% RSLogix 500 project Regelventil Zyklussteuerung.RSS, saved by version 8.30.00.16 %
PROJECT "UNTITLED"    % processor: Bul.1763 MicroLogix 1100 Series B %

PROGRAM FILES
  LAD 2 "MAIN"  4 rungs
  LAD 3 "IO"  7 rungs
  LAD 4 "CONTROL"  31 rungs
  LAD 5 "POSITIONS"  6 rungs

DATA FILES
  O0 OUTPUT  4 elements
  I1 INPUT  6 elements
  S2 STATUS  66 elements
  B3 BINARY  4 elements
  T4 TIMER  3 elements
  C5 COUNTER  1 elements
  R6 CONTROL  1 elements
  N7 INTEGER  3 elements
  F8 FLOAT  1 elements

LADDER 2 "MAIN"
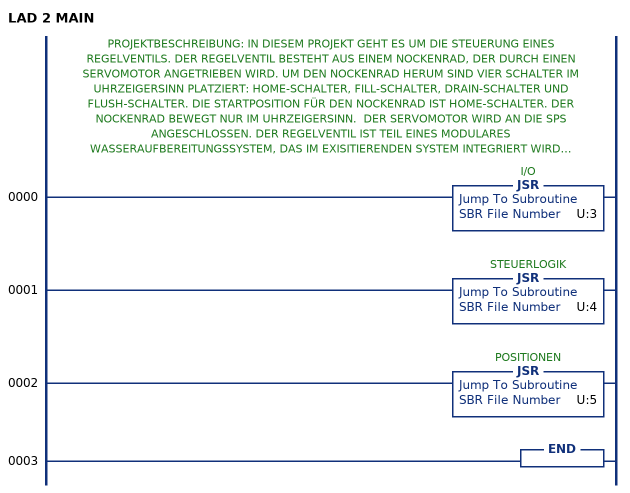
% Rung: 0 %
% PROJEKTBESCHREIBUNG: IN DIESEM PROJEKT GEHT ES UM DIE STEUERUNG EINES REGELVENTILS. DER REGELVENTIL BESTEHT AUS EINEM NOCKENRAD, DER DURCH EINEN SERVOMOTOR ANGETRIEBEN WIRD. UM DEN NOCKENRAD HERUM SIND VIER SCHALTER IM UHRZEIGERSINN PLATZIERT: HOME-SCHALTER, FILL-SCHALTER, DRAIN-SCHALTER UND FLUSH-SCHALTER. DIE STARTPOSITION FÜR DEN NOCKENRAD IST HOME-SCHALTER. DER NOCKENRAD BEWEGT NUR IM UHRZEIGERSINN.  DER SERVOMOTOR WIRD AN DIE SPS ANGESCHLOSSEN. DER REGELVENTIL IST TEIL EINES MODULARES WASSERAUFBEREITUNGSSYSTEM, DAS IM EXISITIERENDEN SYSTEM INTEGRIERT WIRD. DURCH DAS EXISTIERENDE SYSTEM KANN EIN ZYKLUSBEFEHL ERFOLGEN. ANHAND DIESES BEFEHLS WIRD EIN ZYKLUS DURCHGEFÜHRT. DER ZYKLUS DURCHLÄUFT FOLGENDE SCHRITTE:
% 1) FALLS NOCKENRAD SICH NICHT AN STARTPOSITION BEFINDET(HOME-SCHALTER NICHT EINGESCHALTET), DREHT DER NOCKENRAD BIS DER HOME-SCHALTER EINGESCHLATET IST:
% 2) DANN BEWEGT SICH DER NOCKENRAD BIS DER FILL-SCHALTER EINGESCHALTET IST UND DER FILLVORGANG WIRD FÜR 10 SEKUNDEN DURCHGEFÜHRT.
% 3) NACH 10 SEKUNDEN,DER NOCKENRAD BEWEGT SICH WEITER  BIS DER DRAIN-SCHALTER EINGESCHALTET IST. DER DRAINVORGANG WIRD FÜR 20 SEKUNDEN DURCHGEFÜHRT.
% 4) NACH 20 SEKUNDEN, DER NOCKENRAD BEWEGT SICH WEITER BIS DER FLUSH-SCHALTET EINGESCHALTET IST. DER FLUSHVORGAGN WIRD FÜR 10 SEKUNDEN DURCHGEFÜHRT.
% 5) NACH 10 SEKUNDEN, DER NOCKENRAD DREHT SICH WEITER BIS DER HOME-SCHALTET WIEDER EINSCHALTET WIRD. DER ZYKLUS KOMMT ZUM ENDE.
% FERNER HAT DAS PROGRAM DAS INTERRUPT-BIT B3:0/0. FALLS SIE AKTIV WIRD UND DER REGELVENTIL DEN ZYKLUS DURCHLÄUFT, WIRD DER ZYKLUS UNTERBROCHEN UND DER REGELVENTIL KOMMT ZUR STARTPOSITION: %
SOR JSR U:3 EOR
%   U:3  "I/O" %
% Rung: 1 %
SOR JSR U:4 EOR
%   U:4  "STEUERLOGIK" %
% Rung: 2 %
SOR JSR U:5 EOR
%   U:5  "POSITIONEN" %
% Rung: 3 %
SOR END EOR

LADDER 3 "IO"
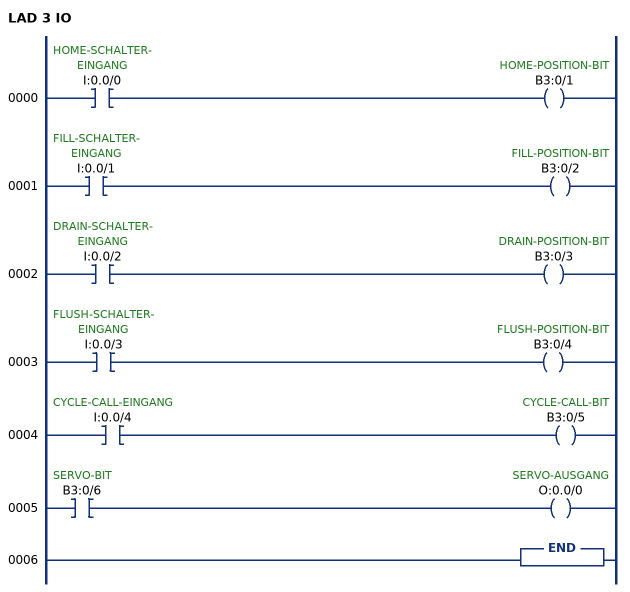
% Rung: 0 %
SOR XIC I:0.0/0 OTE B3:0/1 EOR
%   I:0.0/0  "HOME-SCHALTER- EINGANG" %
%   B3:0/1  "HOME-POSITION-BIT" %
% Rung: 1 %
SOR XIC I:0.0/1 OTE B3:0/2 EOR
%   I:0.0/1  "FILL-SCHALTER- EINGANG" %
%   B3:0/2  "FILL-POSITION-BIT" %
% Rung: 2 %
SOR XIC I:0.0/2 OTE B3:0/3 EOR
%   I:0.0/2  "DRAIN-SCHALTER- EINGANG" %
%   B3:0/3  "DRAIN-POSITION-BIT" %
% Rung: 3 %
SOR XIC I:0.0/3 OTE B3:0/4 EOR
%   I:0.0/3  "FLUSH-SCHALTER- EINGANG" %
%   B3:0/4  "FLUSH-POSITION-BIT" %
% Rung: 4 %
SOR XIC I:0.0/4 OTE B3:0/5 EOR
%   I:0.0/4  "CYCLE-CALL-EINGANG" %
%   B3:0/5  "CYCLE-CALL-BIT" %
% Rung: 5 %
SOR XIC B3:0/6 OTE O:0.0/0 EOR
%   B3:0/6  "SERVO-BIT" %
%   O:0.0/0  "SERVO-AUSGANG" %
% Rung: 6 %
SOR END EOR

LADDER 4 "CONTROL"
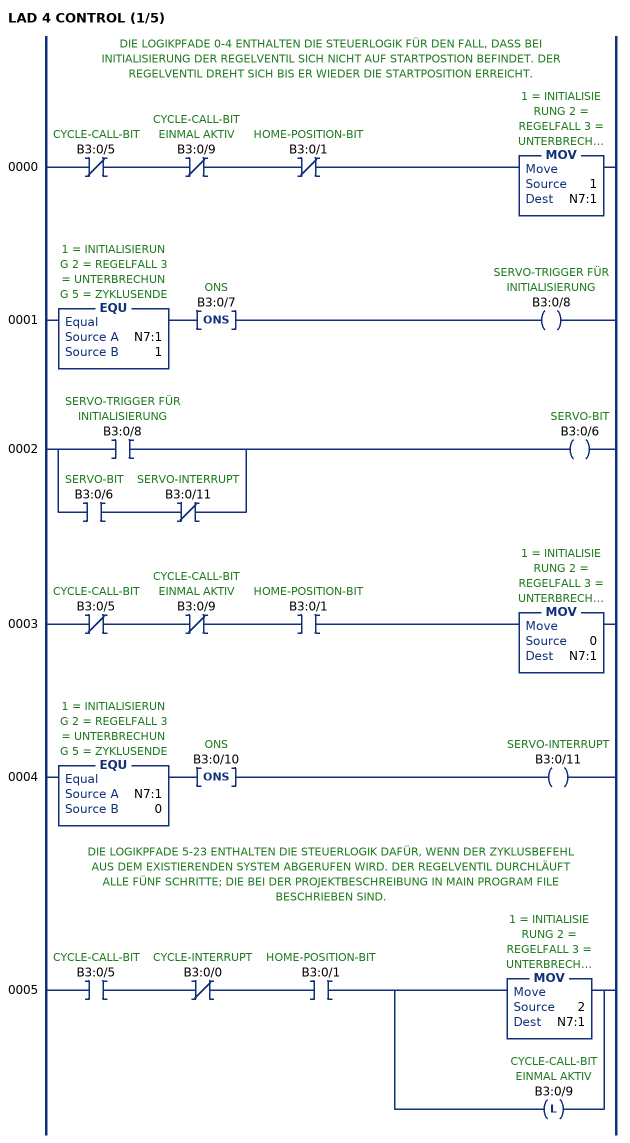
% Rung: 0 %  % edit flag set %
% DIE LOGIKPFADE 0-4 ENTHALTEN DIE STEUERLOGIK FÜR DEN FALL, DASS BEI INITIALISIERUNG DER REGELVENTIL SICH NICHT AUF STARTPOSTION BEFINDET. DER REGELVENTIL DREHT SICH BIS ER WIEDER DIE STARTPOSITION ERREICHT. %
SOR XIO B3:0/5 XIO B3:0/9 XIO B3:0/1 MOV 1 N7:1 EOR
%   B3:0/5  "CYCLE-CALL-BIT" %
%   B3:0/9  "CYCLE-CALL-BIT EINMAL AKTIV" %
%   B3:0/1  "HOME-POSITION-BIT" %
%   N7:1  "1 = INITIALISIERUNG 2 = REGELFALL 3 = UNTERBRECHUNG 5 = ZYKLUSENDE" %
% Rung: 1 %
SOR EQU N7:1 1 ONS B3:0/7 OTE B3:0/8 EOR
%   N7:1  "1 = INITIALISIERUNG 2 = REGELFALL 3 = UNTERBRECHUNG 5 = ZYKLUSENDE" %
%   B3:0/7  "ONS" %
%   B3:0/8  "SERVO-TRIGGER FÜR INITIALISIERUNG" %
% Rung: 2 %
SOR BST XIC B3:0/8 NXB XIC B3:0/6 XIO B3:0/11 BND OTE B3:0/6 EOR
%   B3:0/8  "SERVO-TRIGGER FÜR INITIALISIERUNG" %
%   B3:0/6  "SERVO-BIT" %
%   B3:0/11  "SERVO-INTERRUPT" %
% Rung: 3 %
SOR XIO B3:0/5 XIO B3:0/9 XIC B3:0/1 MOV 0 N7:1 EOR
%   B3:0/5  "CYCLE-CALL-BIT" %
%   B3:0/9  "CYCLE-CALL-BIT EINMAL AKTIV" %
%   B3:0/1  "HOME-POSITION-BIT" %
%   N7:1  "1 = INITIALISIERUNG 2 = REGELFALL 3 = UNTERBRECHUNG 5 = ZYKLUSENDE" %
% Rung: 4 %
SOR EQU N7:1 0 ONS B3:0/10 OTE B3:0/11 EOR
%   N7:1  "1 = INITIALISIERUNG 2 = REGELFALL 3 = UNTERBRECHUNG 5 = ZYKLUSENDE" %
%   B3:0/10  "ONS" %
%   B3:0/11  "SERVO-INTERRUPT" %
% Rung: 5 %
% DIE LOGIKPFADE 5-23 ENTHALTEN DIE STEUERLOGIK DAFÜR, WENN DER ZYKLUSBEFEHL AUS DEM EXISTIERENDEN SYSTEM ABGERUFEN WIRD. DER REGELVENTIL DURCHLÄUFT  ALLE FÜNF SCHRITTE; DIE BEI DER PROJEKTBESCHREIBUNG IN MAIN PROGRAM FILE BESCHRIEBEN SIND. %
SOR XIC B3:0/5 XIO B3:0/0 XIC B3:0/1 BST MOV 2 N7:1 NXB OTL B3:0/9 BND EOR
%   B3:0/5  "CYCLE-CALL-BIT" %
%   B3:0/0  "CYCLE-INTERRUPT" %
%   B3:0/1  "HOME-POSITION-BIT" %
%   N7:1  "1 = INITIALISIERUNG 2 = REGELFALL 3 = UNTERBRECHUNG 5 = ZYKLUSENDE" %
%   B3:0/9  "CYCLE-CALL-BIT EINMAL AKTIV" %

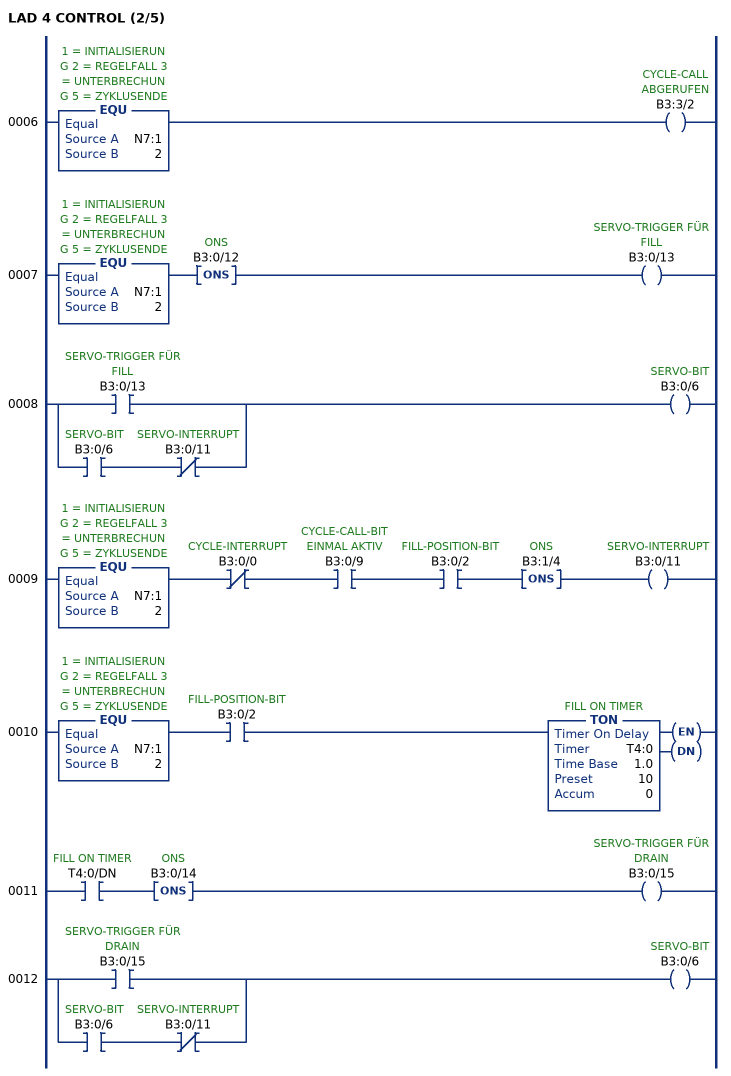
% Rung: 6 %
SOR EQU N7:1 2 OTE B3:3/2 EOR
%   N7:1  "1 = INITIALISIERUNG 2 = REGELFALL 3 = UNTERBRECHUNG 5 = ZYKLUSENDE" %
%   B3:3/2  "CYCLE-CALL ABGERUFEN" %
% Rung: 7 %
SOR EQU N7:1 2 ONS B3:0/12 OTE B3:0/13 EOR
%   N7:1  "1 = INITIALISIERUNG 2 = REGELFALL 3 = UNTERBRECHUNG 5 = ZYKLUSENDE" %
%   B3:0/12  "ONS" %
%   B3:0/13  "SERVO-TRIGGER FÜR FILL" %
% Rung: 8 %
SOR BST XIC B3:0/13 NXB XIC B3:0/6 XIO B3:0/11 BND OTE B3:0/6 EOR
%   B3:0/13  "SERVO-TRIGGER FÜR FILL" %
%   B3:0/6  "SERVO-BIT" %
%   B3:0/11  "SERVO-INTERRUPT" %
% Rung: 9 %
SOR EQU N7:1 2 XIO B3:0/0 XIC B3:0/9 XIC B3:0/2 ONS B3:1/4 OTE B3:0/11 EOR
%   N7:1  "1 = INITIALISIERUNG 2 = REGELFALL 3 = UNTERBRECHUNG 5 = ZYKLUSENDE" %
%   B3:0/0  "CYCLE-INTERRUPT" %
%   B3:0/9  "CYCLE-CALL-BIT EINMAL AKTIV" %
%   B3:0/2  "FILL-POSITION-BIT" %
%   B3:1/4  "ONS" %
%   B3:0/11  "SERVO-INTERRUPT" %
% Rung: 10 %
SOR EQU N7:1 2 XIC B3:0/2 TON T4:0 1.0 10 0 EOR
%   N7:1  "1 = INITIALISIERUNG 2 = REGELFALL 3 = UNTERBRECHUNG 5 = ZYKLUSENDE" %
%   B3:0/2  "FILL-POSITION-BIT" %
%   T4:0  "FILL ON TIMER" %
% Rung: 11 %
SOR XIC T4:0/DN ONS B3:0/14 OTE B3:0/15 EOR
%   T4:0  "FILL ON TIMER" %
%   B3:0/14  "ONS" %
%   B3:0/15  "SERVO-TRIGGER FÜR DRAIN" %
% Rung: 12 %
SOR BST XIC B3:0/15 NXB XIC B3:0/6 XIO B3:0/11 BND OTE B3:0/6 EOR
%   B3:0/15  "SERVO-TRIGGER FÜR DRAIN" %
%   B3:0/6  "SERVO-BIT" %
%   B3:0/11  "SERVO-INTERRUPT" %

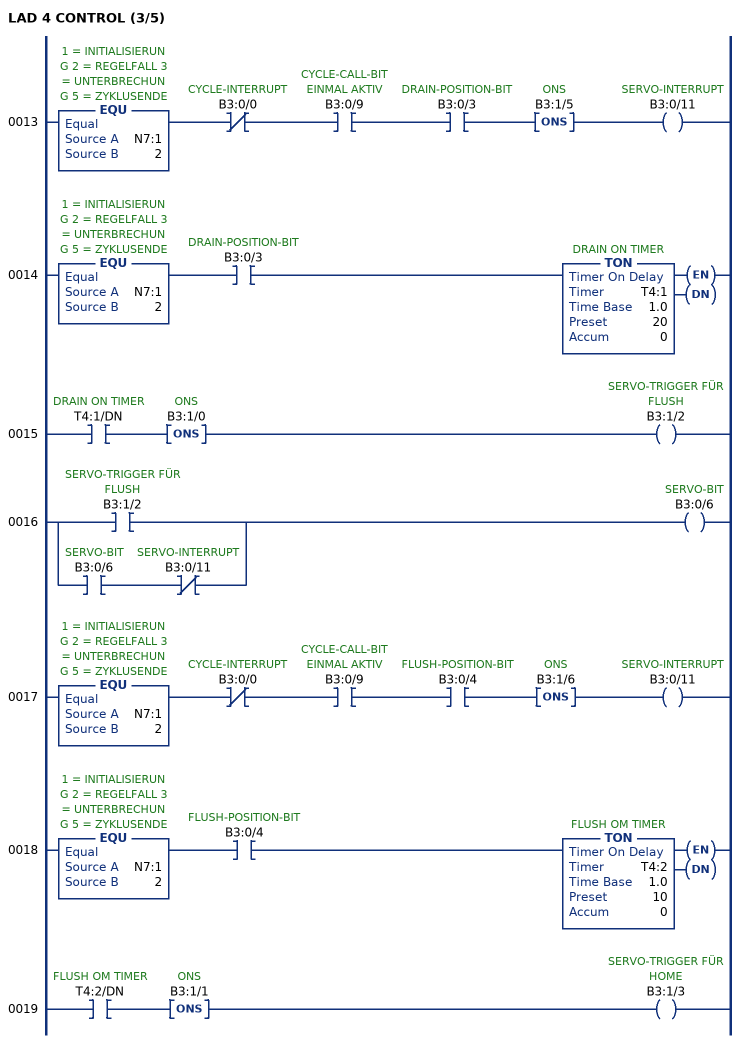
% Rung: 13 %
SOR EQU N7:1 2 XIO B3:0/0 XIC B3:0/9 XIC B3:0/3 ONS B3:1/5 OTE B3:0/11 EOR
%   N7:1  "1 = INITIALISIERUNG 2 = REGELFALL 3 = UNTERBRECHUNG 5 = ZYKLUSENDE" %
%   B3:0/0  "CYCLE-INTERRUPT" %
%   B3:0/9  "CYCLE-CALL-BIT EINMAL AKTIV" %
%   B3:0/3  "DRAIN-POSITION-BIT" %
%   B3:1/5  "ONS" %
%   B3:0/11  "SERVO-INTERRUPT" %
% Rung: 14 %
SOR EQU N7:1 2 XIC B3:0/3 TON T4:1 1.0 20 0 EOR
%   N7:1  "1 = INITIALISIERUNG 2 = REGELFALL 3 = UNTERBRECHUNG 5 = ZYKLUSENDE" %
%   B3:0/3  "DRAIN-POSITION-BIT" %
%   T4:1  "DRAIN ON TIMER" %
% Rung: 15 %
SOR XIC T4:1/DN ONS B3:1/0 OTE B3:1/2 EOR
%   T4:1  "DRAIN ON TIMER" %
%   B3:1/0  "ONS" %
%   B3:1/2  "SERVO-TRIGGER FÜR FLUSH" %
% Rung: 16 %
SOR BST XIC B3:1/2 NXB XIC B3:0/6 XIO B3:0/11 BND OTE B3:0/6 EOR
%   B3:1/2  "SERVO-TRIGGER FÜR FLUSH" %
%   B3:0/6  "SERVO-BIT" %
%   B3:0/11  "SERVO-INTERRUPT" %
% Rung: 17 %
SOR EQU N7:1 2 XIO B3:0/0 XIC B3:0/9 XIC B3:0/4 ONS B3:1/6 OTE B3:0/11 EOR
%   N7:1  "1 = INITIALISIERUNG 2 = REGELFALL 3 = UNTERBRECHUNG 5 = ZYKLUSENDE" %
%   B3:0/0  "CYCLE-INTERRUPT" %
%   B3:0/9  "CYCLE-CALL-BIT EINMAL AKTIV" %
%   B3:0/4  "FLUSH-POSITION-BIT" %
%   B3:1/6  "ONS" %
%   B3:0/11  "SERVO-INTERRUPT" %
% Rung: 18 %
SOR EQU N7:1 2 XIC B3:0/4 TON T4:2 1.0 10 0 EOR
%   N7:1  "1 = INITIALISIERUNG 2 = REGELFALL 3 = UNTERBRECHUNG 5 = ZYKLUSENDE" %
%   B3:0/4  "FLUSH-POSITION-BIT" %
%   T4:2  "FLUSH OM TIMER" %
% Rung: 19 %
SOR XIC T4:2/DN ONS B3:1/1 OTE B3:1/3 EOR
%   T4:2  "FLUSH OM TIMER" %
%   B3:1/1  "ONS" %
%   B3:1/3  "SERVO-TRIGGER FÜR HOME" %

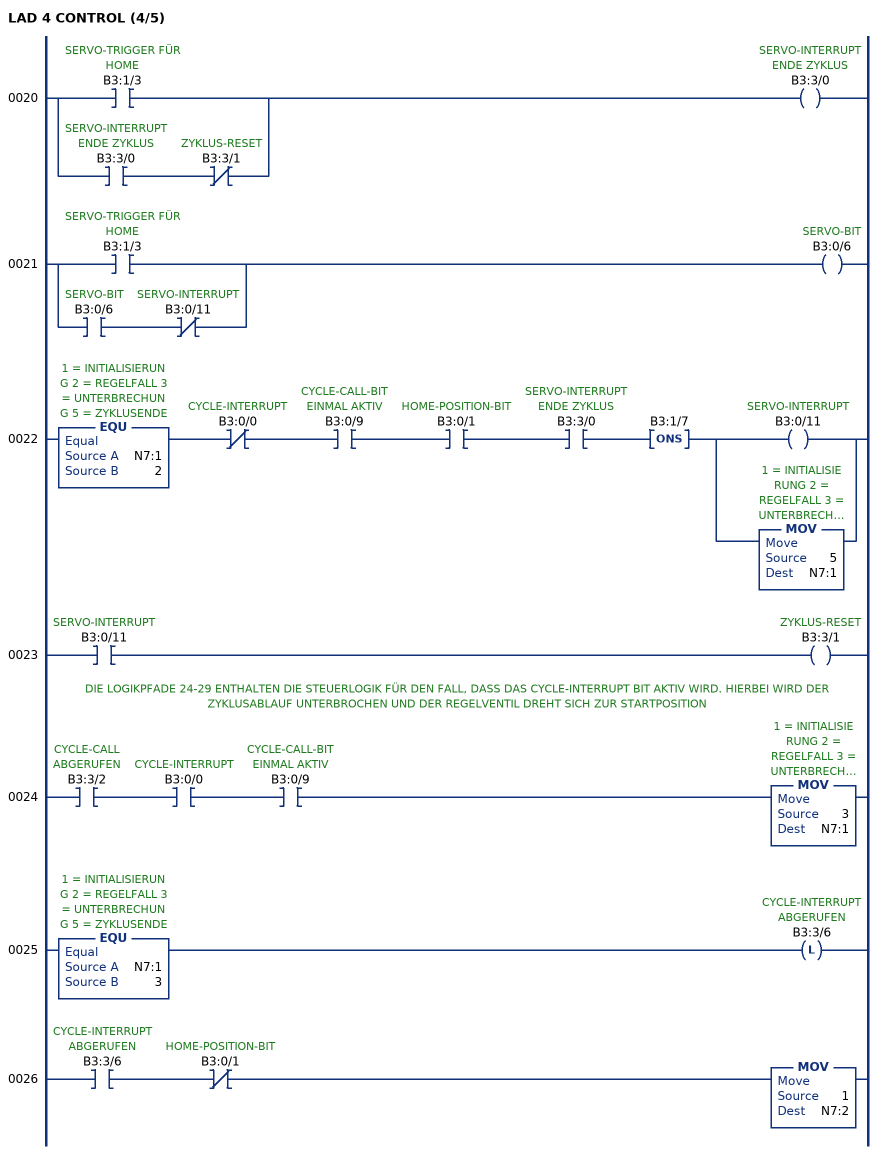
% Rung: 20 %
SOR BST XIC B3:1/3 NXB XIC B3:3/0 XIO B3:3/1 BND OTE B3:3/0 EOR
%   B3:1/3  "SERVO-TRIGGER FÜR HOME" %
%   B3:3/0  "SERVO-INTERRUPT ENDE ZYKLUS" %
%   B3:3/1  "ZYKLUS-RESET" %
% Rung: 21 %
SOR BST XIC B3:1/3 NXB XIC B3:0/6 XIO B3:0/11 BND OTE B3:0/6 EOR
%   B3:1/3  "SERVO-TRIGGER FÜR HOME" %
%   B3:0/6  "SERVO-BIT" %
%   B3:0/11  "SERVO-INTERRUPT" %
% Rung: 22 %
SOR EQU N7:1 2 XIO B3:0/0 XIC B3:0/9 XIC B3:0/1 XIC B3:3/0 ONS B3:1/7 BST OTE B3:0/11 NXB MOV 5 N7:1 BND EOR
%   N7:1  "1 = INITIALISIERUNG 2 = REGELFALL 3 = UNTERBRECHUNG 5 = ZYKLUSENDE" %
%   B3:0/0  "CYCLE-INTERRUPT" %
%   B3:0/9  "CYCLE-CALL-BIT EINMAL AKTIV" %
%   B3:0/1  "HOME-POSITION-BIT" %
%   B3:3/0  "SERVO-INTERRUPT ENDE ZYKLUS" %
%   B3:0/11  "SERVO-INTERRUPT" %
% Rung: 23 %
SOR XIC B3:0/11 OTE B3:3/1 EOR
%   B3:0/11  "SERVO-INTERRUPT" %
%   B3:3/1  "ZYKLUS-RESET" %
% Rung: 24 %
% DIE LOGIKPFADE 24-29 ENTHALTEN DIE STEUERLOGIK FÜR DEN FALL, DASS DAS CYCLE-INTERRUPT BIT AKTIV WIRD. HIERBEI WIRD DER ZYKLUSABLAUF UNTERBROCHEN UND DER REGELVENTIL DREHT SICH ZUR STARTPOSITION %
SOR XIC B3:3/2 XIC B3:0/0 XIC B3:0/9 MOV 3 N7:1 EOR
%   B3:3/2  "CYCLE-CALL ABGERUFEN" %
%   B3:0/0  "CYCLE-INTERRUPT" %
%   B3:0/9  "CYCLE-CALL-BIT EINMAL AKTIV" %
%   N7:1  "1 = INITIALISIERUNG 2 = REGELFALL 3 = UNTERBRECHUNG 5 = ZYKLUSENDE" %
% Rung: 25 %
SOR EQU N7:1 3 OTL B3:3/6 EOR
%   N7:1  "1 = INITIALISIERUNG 2 = REGELFALL 3 = UNTERBRECHUNG 5 = ZYKLUSENDE" %
%   B3:3/6  "CYCLE-INTERRUPT ABGERUFEN" %
% Rung: 26 %
SOR XIC B3:3/6 XIO B3:0/1 MOV 1 N7:2 EOR
%   B3:3/6  "CYCLE-INTERRUPT ABGERUFEN" %
%   B3:0/1  "HOME-POSITION-BIT" %

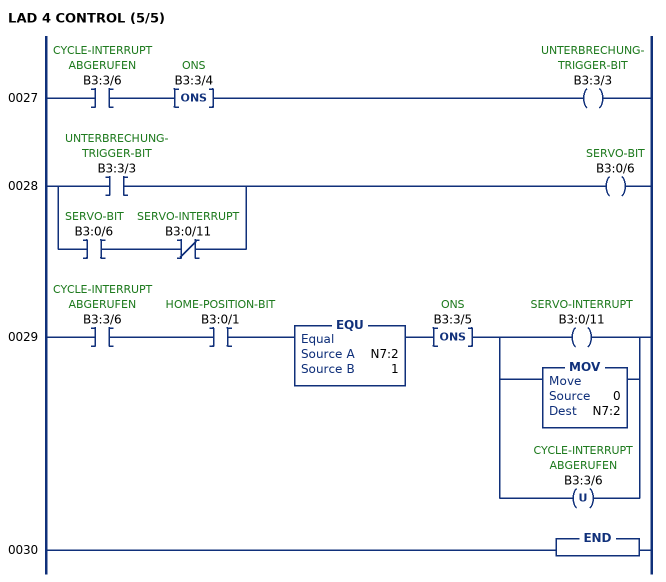
% Rung: 27 %
SOR XIC B3:3/6 ONS B3:3/4 OTE B3:3/3 EOR
%   B3:3/6  "CYCLE-INTERRUPT ABGERUFEN" %
%   B3:3/4  "ONS" %
%   B3:3/3  "UNTERBRECHUNG- TRIGGER-BIT" %
% Rung: 28 %
SOR BST XIC B3:3/3 NXB XIC B3:0/6 XIO B3:0/11 BND OTE B3:0/6 EOR
%   B3:3/3  "UNTERBRECHUNG- TRIGGER-BIT" %
%   B3:0/6  "SERVO-BIT" %
%   B3:0/11  "SERVO-INTERRUPT" %
% Rung: 29 %
SOR XIC B3:3/6 XIC B3:0/1 EQU N7:2 1 ONS B3:3/5 BST OTE B3:0/11 NXB MOV 0 N7:2 NXB OTU B3:3/6 BND EOR
%   B3:3/6  "CYCLE-INTERRUPT ABGERUFEN" %
%   B3:0/1  "HOME-POSITION-BIT" %
%   B3:3/5  "ONS" %
%   B3:0/11  "SERVO-INTERRUPT" %
% Rung: 30 %
SOR END EOR

LADDER 5 "POSITIONS"
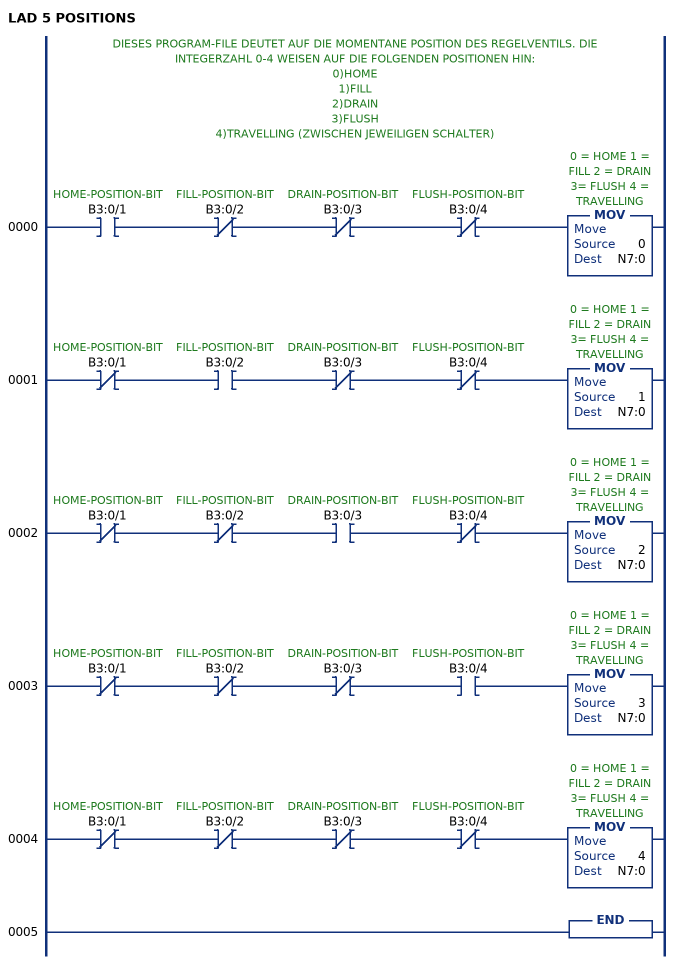
% Rung: 0 %
% DIESES PROGRAM-FILE DEUTET AUF DIE MOMENTANE POSITION DES REGELVENTILS. DIE INTEGERZAHL 0-4 WEISEN AUF DIE FOLGENDEN POSITIONEN HIN:
% 0)HOME
% 1)FILL
% 2)DRAIN
% 3)FLUSH
% 4)TRAVELLING (ZWISCHEN JEWEILIGEN SCHALTER) %
SOR XIC B3:0/1 XIO B3:0/2 XIO B3:0/3 XIO B3:0/4 MOV 0 N7:0 EOR
%   B3:0/1  "HOME-POSITION-BIT" %
%   B3:0/2  "FILL-POSITION-BIT" %
%   B3:0/3  "DRAIN-POSITION-BIT" %
%   B3:0/4  "FLUSH-POSITION-BIT" %
%   N7:0  "0 = HOME 1 = FILL 2 = DRAIN 3= FLUSH 4 = TRAVELLING" %
% Rung: 1 %
SOR XIO B3:0/1 XIC B3:0/2 XIO B3:0/3 XIO B3:0/4 MOV 1 N7:0 EOR
%   B3:0/1  "HOME-POSITION-BIT" %
%   B3:0/2  "FILL-POSITION-BIT" %
%   B3:0/3  "DRAIN-POSITION-BIT" %
%   B3:0/4  "FLUSH-POSITION-BIT" %
%   N7:0  "0 = HOME 1 = FILL 2 = DRAIN 3= FLUSH 4 = TRAVELLING" %
% Rung: 2 %
SOR XIO B3:0/1 XIO B3:0/2 XIC B3:0/3 XIO B3:0/4 MOV 2 N7:0 EOR
%   B3:0/1  "HOME-POSITION-BIT" %
%   B3:0/2  "FILL-POSITION-BIT" %
%   B3:0/3  "DRAIN-POSITION-BIT" %
%   B3:0/4  "FLUSH-POSITION-BIT" %
%   N7:0  "0 = HOME 1 = FILL 2 = DRAIN 3= FLUSH 4 = TRAVELLING" %
% Rung: 3 %
SOR XIO B3:0/1 XIO B3:0/2 XIO B3:0/3 XIC B3:0/4 MOV 3 N7:0 EOR
%   B3:0/1  "HOME-POSITION-BIT" %
%   B3:0/2  "FILL-POSITION-BIT" %
%   B3:0/3  "DRAIN-POSITION-BIT" %
%   B3:0/4  "FLUSH-POSITION-BIT" %
%   N7:0  "0 = HOME 1 = FILL 2 = DRAIN 3= FLUSH 4 = TRAVELLING" %
% Rung: 4 %
SOR XIO B3:0/1 XIO B3:0/2 XIO B3:0/3 XIO B3:0/4 MOV 4 N7:0 EOR
%   B3:0/1  "HOME-POSITION-BIT" %
%   B3:0/2  "FILL-POSITION-BIT" %
%   B3:0/3  "DRAIN-POSITION-BIT" %
%   B3:0/4  "FLUSH-POSITION-BIT" %
%   N7:0  "0 = HOME 1 = FILL 2 = DRAIN 3= FLUSH 4 = TRAVELLING" %
% Rung: 5 %
SOR END EOR

OTHER DOCUMENTED ADDRESSES
  B3:1/8  "SERVO-TRIGGER-BIT- FÜR DRAIN"
  B3:1/9  "SERVO-TRIGGER-BIT- FÜR FLUSH"
  B3:1/10  "SERVO-TRIGGER-BIT- FÜR HOME"
  B3:1/11  "SERVO-TRIGGER-BIT FÜR INTERRUPT"
  B3:1/12  "SERVO-TRIGGER-BIT FÜR INITIALISIERUNG"
  B3:2/0  "INITIALISIERUNGBIT"
  B3:3/7  "STORAGE BIT"
  U:6  "REGELFALL"
  U:7  "UNTERBRECHUNG"
  U:8  "SONDERFALL"
  U:9  "INITIALISIERUNG"

DATA TABLE (non-zero values as saved)
DATA T4
% .PRE .ACC %
% T4:0 % 10 0
% T4:1 % 20 0
% T4:2 % 10 0
